// TIA Portal project "Hugo_Uriel_Travail_1" (V19)

(* hardware
DEVICE "HMI_1"  KTP700 Basic PN
   slot 0: "HMI_1"  KTP700 Basic PN  6AV2 123-2GB03-0AX0  17.0.0.0
   slot 1: "HMI_RT_1"  KTP700 Basic PN  6AV2 123-2GB03-0AX0  17.0.0.0
   slot 5: "HMI_1.IE_CP_1"  PROFINET Interface  17.0.0.0
      slot 1: "PROFINET Interface_1"  PROFINET Interface
         slot 1: "Port_1"  Port
DEVICE "S7-300/ET200M station_1"  S7-300 station
   slot 0: "Rail_0"  Rail  6ES7 390-1***0-0AA0
   slot 2: "PLC_1"  CPU 314C-2 PN/DP  6ES7 314-6EH04-0AB0  V3.3
      slot 2: "PROFINET interface_1"  PN-IO
         slot 1: "Port_1"  Port
         slot 2: "Port_2"  Port
      slot 5: "DI 24/DO 16_1"  DI24/DO16
      slot 6: "AI 5/AO 2_1"  AI5/AO2
      slot 7: "Count_1"  Counter
      slot 8: "Positioning_1"  Positioning
*)

// ===== PLC "PLC_1"  CPU 314C-2 PN/DP =====

VAR_GLOBAL   // PLC tag table "Default tag table"
   "Memoire pièce haute HMI" AT %M50.0 : Bool;
   "Memoire pièce basse HMI" AT %M50.1 : Bool;
   "Memoire pas de pièce HMI" AT %M50.2 : Bool;
   "Memoire B5" AT %M50.3 : Bool;
   "Memoire B6" AT %M50.4 : Bool;
   "HMI_M1" AT %M50.5 : Bool;
   "HMI_M2" AT %M50.6 : Bool;
   "HMI_1M1" AT %M50.7 : Bool;
   "HMI_2M1" AT %M51.0 : Bool;
END_VAR

VAR_GLOBAL   // PLC tag table "Variables Station Separating"
   "PART_AV" AT %I0.0 : Bool;   // Pièce Disponible
   "B2" AT %I0.1 : Bool;   // Présence pièce pour analyxe
   "B3" AT %I0.2 : Bool;   // Vérification profondeur pièce
   "B4" AT %I0.3 : Bool;   // Vérin rotatif rentré
   "B5" AT %I0.4 : Bool;   // Convoyeur 2 plein
   "B6" AT %I0.5 : Bool;   // Pièce en sortie de station
   "IP_FI_B" AT %I0.6 : Bool;   // Simulation station suivante libre
   "IP_FI" AT %I0.7 : Bool;   // Station suivante libre
   "BP Start" AT %I1.0 : Bool;   // NO Départ cycle
   "BP Stop" AT %I1.1 : Bool;   // NF Fin cycle
   "Selecteur Auto/Manu" AT %I1.2 : Bool;   // Choix mode fonctionnement
   "BP Reset" AT %I1.3 : Bool;   // Initialisation station
   "Emergency Stop" AT %I1.5 : Bool;   // Arrêt d'urgence (ponté)
   "M1" AT %Q0.0 : Bool;   // Convoyeur principal - Marche
   "M2" AT %Q0.1 : Bool;   // Convoyeur secondaire - Marche
   "1M1" AT %Q0.2 : Bool;   // Blocage pièce - sorti au repos
   "2M1" AT %Q0.3 : Bool;   // Aiguillage - convoyeur secondaire
   "IP_N_FO" AT %Q0.7 : Bool;   // Station occupée
   "LStart" AT %Q1.0 : Bool;   // Lampe BP Start
   "LReset" AT %Q1.1 : Bool;   // Lampe BP Reset
   "Q1" AT %Q1.2 : Bool;   // Voyant lumineux Gauche
   "Q2" AT %Q1.3 : Bool;   // Voyant lumineux Droite
   "B3 Analogique" AT %IW800 : Int;   // Profondeur Pièce
END_VAR

VAR_GLOBAL   // PLC tag table "Memoires"
   "FP0" AT %M30.0 : Bool;
   "FN0" AT %M31.0 : Bool;
   "FP1" AT %M30.1 : Bool;
   "FN1" AT %M31.1 : Bool;
   "Memoire_TP_Mesure" AT %M32.0 : Bool;
   "Memoire_TP_B5" AT %M32.1 : Bool;
   "RET_VAL" AT %MW10 : Word;
   "Sortie_Scale" AT %MD20 : Real;
   "Scale_bipolaire" AT %M33.0 : Bool;
   "FP2" AT %M30.2 : Bool;
   "FN2" AT %M31.2 : Bool;
   "FN3" AT %M31.3 : Bool;
   "Memoire_TP_B5_result" AT %M33.1 : Bool;
END_VAR

DATA_BLOCK "Tapis_roulant_DB_2"   // DB3
{ S7_Optimized_Access := 'FALSE' }
VERSION : 0.1
// stored: InstanceOfName Tapis_roulant_DB
"Tapis_roulant_DB"
BEGIN
END_DATA_BLOCK

DATA_BLOCK "Verrin_DB_Aiguillage"   // DB4
{ S7_Optimized_Access := 'FALSE' }
VERSION : 0.1
// stored: InstanceOfName Verrin_DB
"Verrin_DB"
BEGIN
END_DATA_BLOCK

DATA_BLOCK "Verrin_DB_blocage"   // DB5
{ S7_Optimized_Access := 'FALSE' }
VERSION : 0.1
// stored: InstanceOfName Verrin_DB
"Verrin_DB"
BEGIN
END_DATA_BLOCK

DATA_BLOCK "Data_block_memo"   // DB8
{ S7_Optimized_Access := 'FALSE' }
VERSION : 0.1
   VAR
      memo_convoyeur_1 : Bool;
      memo_convoyeur_2 : Bool;
      memo_verrin_aiguillage : Bool;
      memo_verrin_blocage : Bool;
      IN_Avancer_Tapis_1 : Bool;
      IN_Avancer_Tapis_2 : Bool;
      IN_Verrin_blocage : Bool;
      IN_Verrin_aiguillage : Bool;
      OUT_position_verrin_aiguillage : Bool;
      OUT_position_verrin_blocage : Bool;
      valeur_profondeur : Real;
      rent_val_capteur : Word;
      auto : Bool;
      manu : Bool;
      marche : Bool;
      arret : Bool;
      STATE : Int;
      profondeur : Bool;
   END_VAR
BEGIN
END_DATA_BLOCK

DATA_BLOCK "Tapis_roulant_DB_1"   // DB9
{ S7_Optimized_Access := 'FALSE' }
VERSION : 0.1
// stored: InstanceOfName Tapis_roulant_DB
"Tapis_roulant_DB"
BEGIN
END_DATA_BLOCK

DATA_BLOCK "Grafcet_DB"   // DB10
{ S7_Optimized_Access := 'FALSE' }
VERSION : 0.1
// stored: InstanceOfName Grafcet
"Grafcet"
BEGIN
END_DATA_BLOCK

FUNCTION_BLOCK "Verrin_DB"   // FB1, FBD
{ S7_Optimized_Access := 'FALSE' }
VERSION : 0.1
   VAR_INPUT
      Activation : Bool;
      Positon : Bool;
   END_VAR
   VAR_OUTPUT
      Marche : Bool;
      Position_retour : Bool;
   END_VAR
BEGIN

REGION Network 1
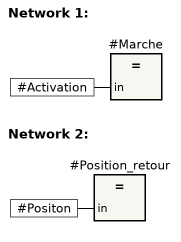
   #Marche := #Activation;
END_REGION

REGION Network 2
   #Position_retour := #Positon;
END_REGION
END_FUNCTION_BLOCK

FUNCTION_BLOCK "Tapis_roulant_DB"   // FB2, FBD
{ S7_Optimized_Access := 'FALSE' }
VERSION : 0.1
   VAR_INPUT
      Start_Avant : Bool;
   END_VAR
   VAR_OUTPUT
      Run : Bool;
   END_VAR
   VAR_TEMP
      moteur_tapis : Bool;
   END_VAR
BEGIN

REGION Network 1
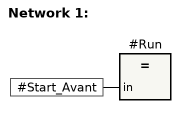
   #Run := #Start_Avant;
END_REGION
END_FUNCTION_BLOCK

FUNCTION_BLOCK "Grafcet"   // FB3, GRAPH
{ S7_Optimized_Access := 'FALSE' }
VERSION : 0.1
   VAR_INPUT
      OFF_SQ : Bool := false;   // Turn sequence off
      INIT_SQ : Bool := false;   // Set sequence to initial state
      ACK_EF : Bool := false;   // Acknowledge all errors and faults
      S_PREV : Bool := false;   // Output previous step in parameter S_NO
      S_NEXT : Bool := false;   // Indicate next step in parameter S_NO
      SW_AUTO : Bool := false;   // Automatic mode
      SW_TAP : Bool := false;   // Semiautomatic/switch with transition
      SW_TOP : Bool := false;   // Semiautomatic/ignore transition
      SW_MAN : Bool := false;   // Manual mode
      S_SEL : Int := 0;   // Select step to be output to S_NO
      S_ON : Bool := false;   // Activate step indicated in S_NO
      S_OFF : Bool := false;   // Disable step indicated in S_NO
      T_PUSH : Bool := false;   // Enable transition to switch in semi automatic mode
   END_VAR
   VAR_OUTPUT
      S_NO : Int := 0;   // Step number
      S_MORE : Bool := false;   // More steps are available and can be shown in S_NO
      S_ACTIVE : Bool := false;   // Step indicated in S_NO is active
      ERR_FLT : Bool := false;   // Interlock or supervision group error
      AUTO_ON : Bool := false;   // Automatic mode is active
      TAP_ON : Bool := false;   // Semiautomatic mode/step with transition enabled
      TOP_ON : Bool := false;   // Semiautomatic mode/ignore transition enabled
      MAN_ON : Bool := false;   // Manual mode is active
   END_VAR
   VAR
      SWITCH : Array[0..0] of DWord;
      SW_SQTS : Array[0..9] of Byte;
      SW_ADDR : Word := 16#A;
      G7T_0 : GraphTransition;
      G7S_0 : GraphStep;
      PRE_CRIT : Array[0..0] of DWord;
      POST_CRIT : Array[0..0] of DWord;
      TVX : Array[0..6] of Byte;
      TTX : Array[0..6] of Byte;
      TSX : Array[0..2] of Byte;
      S00X : Array[0..2] of Byte;
      SOFFX : Array[0..2] of Byte;
      SONX : Array[0..2] of Byte;
      SAX : Array[0..2] of Byte;
      SERRX : Array[0..10] of Byte;
      SMX : Array[0..10] of Byte;
      S0X : Array[0..10] of Byte;
      S1X : Array[0..10] of Byte;
      S_DISPLAY : Int;   // Internal display of output parameter S_NO
      S_SEL_OLD : Int;   // Previous value in S_SEL
      S_DISPIDX : Byte;   // Index of the step in S_NO
      T_DISPIDX : Byte;   // Index of the transition displayed in T_NO
      MOPEDGE : Struct
         AUTO : Bool := false;
         MAN : Bool := false;
         TAP : Bool := false;
         TOP : Bool := false;
         ACK_S : Bool := false;
         REG_S : Bool := false;
         T_PREV : Bool := false;
         T_NEXT : Bool := false;
         LOCK : Bool := false;
         SUP : Bool := false;
         ACKREQ : Bool := false;
         SSKIP : Bool := false;
         OFF : Bool := false;
         INIT : Bool := false;
         HALT : Bool := false;
         TMS_HALT : Bool := false;
         OPS_ZERO : Bool := false;
         SACT_DISP : Bool := false;
         SEF_DISP : Bool := false;
         SALL_DISP : Bool := false;
         S_PREV : Bool := false;
         S_NEXT : Bool := false;
         S_SELOK : Bool := false;
         S_ON : Bool := false;
         S_OFF : Bool := false;
         T_PUSH : Bool := false;
         REG : Bool := false;
         ACK : Bool := false;
         IL_PERM : Bool := false;
         T_PERM : Bool := false;
         ILP_MAN : Bool := false;
      END_STRUCT;
      MOP : Struct   // Mode
         AUTO : Bool := true;   // Status: automatic mode
         MAN : Bool := false;   // Status: manual mode
         TAP : Bool := false;   // Status: semi automatic/switch with transition
         TOP : Bool := false;   // Status: semi automatic/ignore transition
         ACK_S : Bool := false;   // Request: acknowledge step at parameter S_NO
         REG_S : Bool := false;   // Request: register step indicated in S_NO
         T_PREV : Bool := false;   // Request: output previous valid transition in T_NO
         T_NEXT : Bool := false;   // Request: output next valid transition in T_NO
         LOCK : Bool := true;   // Status: interlocks enabled
         SUP : Bool := true;   // Status: supervisions enabled
         ACKREQ : Bool := true;   // Status: acknowledgment required
         SSKIP : Bool := false;   // Status: "Skip steps" enabled
         OFF : Bool := false;   // Request: deactivate all steps
         INIT : Bool := true;   // Request: set sequence to initial state
         HALT : Bool := false;   // Status: sequence halted
         TMS_HALT : Bool := false;   // Status: all internal timers held
         OPS_ZERO : Bool := false;   // Status: set all operands processed with N, L, D instructions to 0
         SACT_DISP : Bool := true;   // Status: display active steps only
         SEF_DISP : Bool := false;   // Status: display only steps with errors and disrupted steps
         SALL_DISP : Bool := false;   // Status: display all steps
         S_PREV : Bool := false;   // Request: output previous step to S_NO
         S_NEXT : Bool := false;   // Request: Output next step at S_NO parameter
         S_SELOK : Bool := false;   // Request: output step number from S_SEL to S_NO
         S_ON : Bool := false;   // Request: activate step indicated in S_NO
         S_OFF : Bool := false;   // Request: deactivate step at parameter S_NO
         T_PUSH : Bool := false;   // Request: transition switching enabled
         REG : Bool := false;   // Request: register all interlock and supervision errors
         ACK : Bool := false;   // Request: acknowledge all interlock and supervision errors
         IL_PERM : Bool := false;   // Status: permanent processing of all interlocks
         T_PERM : Bool := false;   // Status: permanent processing of all transitions
         ILP_MAN : Bool := false;   // Status: permanent processing of all interlocks in manual mode
      END_STRUCT;
      TICKS : Struct   // Clock speeds
         DELTA : Time := T#0ms;   // Time difference between two cycles
         OLD : Time := T#0ms;   // 10 ms clock counter value in last cycle
         NEW : Time := T#0ms;   // 10 ms clock counter value in this cycle
      END_STRUCT;
      SQ_FLAGS : Struct   // Sequence bit memory
         ERR_FLT : Bool := false;   // Interlock and supervision group error
         ERROR : Bool := false;   // Interlock group error
         FAULT : Bool := false;   // Supervision group error
         RT_FAIL : Bool := false;   // Runtime error
         NO_SNO : Bool := false;   // Requested step number not found
         NF_OFL : Bool := false;   // Overflow: too many ON or OFF requests
         SA_OFL : Bool := false;   // Overflow: too many steps active
         TV_OFL : Bool := false;   // Overflow: too many valid transitions
         MSG_OFL : Bool := false;   // Overflow: not enough system resources for ALARM_S
         NO_SWI : Bool := false;   // Do not switch in this cycle
         CYC_OP : Bool := false;   // Cyclic execution of the sequence after initialization
         AS_MSG : Bool := true;   // Alarms during runtime enabled or disabled by instruction
         AS_SEND : Bool := false;   // Send alarms from WR_USMSG or only enter in diagnostics buffer
         SQ_BUSY : Bool := false;   // Internal edge bit memory for sequence processing
         SA_BUSY : Bool := false;   // Internal edge bit memory for sequence processing
         AS_SIG : Bool := false;   // Edge bit memory for alarms from Alarm_S and Alarm_SQ
      END_STRUCT;
      S_PTR : DWord := 16#6D0;
      S_PTR2 : DWord := 16#0;
      S_PTR3 : DWord := 16#1350;
      S_PTR4 : DWord := 16#12F0;
      T_PTR : DWord := 16#1290;
      C_AR2 : DWord := 16#0;
      M_FBDB : DWord := 16#30000;
      M_SNO : Word := 16#0;
      M_EVID : Word := 16#0;
      M_EVIL : C_Alarm_s;
      M_EVSV : C_Alarm_s;
      M_EV : DWord := 16#11D0;
      CRIT : Array[0..31] of Bool;
      S_START : Byte := 16#0;
      S_IDX : Byte := 16#0;
      S_INT : Int := 72;
      S_TMP : Byte := 16#0;
      T_START : Byte := 16#0;
      T_IDX : Byte := 16#0;
      T_TMP : Byte := 16#0;
      T_TMP2 : Byte := 16#00;
      TV_POT : Byte := 16#06;
      RETURN1 : Byte := 16#0;
      RETURN2 : Byte := 16#0;
      SINI : Array[0..2] of Byte;
      LSTT : Array[0..11] of Byte;
      ATAJ : Array[0..11] of Byte;
      ATAB : Array[0..11] of Byte;
      PSTT : Array[0..11] of Byte;
      NSTT : Array[0..11] of Byte;
      ASSJ : Array[0..9] of Byte;
      ASSB : Array[0..9] of Byte;
      PTTS : Array[0..9] of Byte;
      NTTS : Array[0..9] of Byte;
      PRE_CNT : Word := 16#1;
      POST_CNT : Word := 16#1;
      ADR_COND : Word := 16#0;
      MAX_TVAL : Byte := 16#5;
      MAX_SACT : Byte := 16#1;
      MAX_CRIT : Byte := 16#4;
      T_CNT : Byte := 16#B;
      SUP_CNT : Byte := 16#0;
      LOCK_CNT : Byte := 16#0;
      S_CNT : Byte := 16#9;
      SQ_CNT : Byte := 16#1;
      PRS_INPAR : DWord := 16#E000FEC8;
      PRS_OUTPAR : DWord := 16#E000800F;
      GC_FLAGS : Struct
         T_MACH : Byte := 16#EB;
         COND_ED : Byte := 16#E3;
         W_LEVEL : Byte := 16#D5;
         FB_IF : Byte := 16#FA;
         AS_MSG : Word := 16#404;
         SSB : Word := 16#108;
         DILG : Word := 16#35E;
         ADDR_T0 : Word := 16#1A;
         CRIT_AVAIL : Bool := false;
         SSKIP_AVAIL : Bool := true;
         SSKIP_ON : Bool := false;
         ACK_REQ : Bool := true;
         SYNC_AVAIL : Bool := true;
         ILP_MAN : Bool := false;
         SWM_LOCKED : Bool := false;
         SAVE_SW : Bool := true;
      END_STRUCT;
      G7_FBMARK : Byte := 16#3C;
      G7_RELEASE : Byte := 16#3C;
      G7_ID2 : Byte := 16#37;
      G7_ID1 : Byte := 16#47;
   END_VAR
   // SW_SQTS[0] := 16#5;
   // SW_SQTS[5] := 16#2;
   // SW_SQTS[4] := 16#1;
   // SW_SQTS[3] := 16#1;
   // SW_SQTS[6] := 16#2;
   // SW_SQTS[7] := 16#3;
   // SW_SQTS[8] := 16#3;
   // SW_SQTS[9] := 16#4;
   // TVX[0] := 16#1;
   // TTX[0] := 16#1;
   // TSX[0] := 16#1;
   // S00X[0] := 16#1;
   // SOFFX[0] := 16#1;
   // SONX[0] := 16#1;
   // SAX[0] := 16#1;
   // SERRX[0] := 16#1;
   // SMX[0] := 16#1;
   // S0X[0] := 16#1;
   // S1X[0] := 16#1;
   // SINI[0] := 16#2;
   // SINI[1] := 16#1;
   // SINI[2] := 0;
   // LSTT[0] := 0;
   // LSTT[1] := 0;
   // LSTT[2] := 0;
   // LSTT[3] := 0;
   // LSTT[4] := 0;
   // LSTT[5] := 0;
   // LSTT[6] := 0;
   // LSTT[7] := 16#3;
   // LSTT[8] := 0;
   // LSTT[9] := 0;
   // LSTT[10] := 16#3;
   // LSTT[11] := 16#2;
   // ATAJ[0] := 0;
   // ATAJ[1] := 16#1;
   // ATAJ[2] := 16#2;
   // ATAJ[3] := 16#3;
   // ATAJ[4] := 16#4;
   // ATAJ[5] := 16#5;
   // ATAJ[6] := 16#6;
   // ATAJ[7] := 16#7;
   // ATAJ[8] := 16#8;
   // ATAJ[9] := 16#9;
   // ATAJ[10] := 16#A;
   // ATAJ[11] := 16#B;
   // ATAB[0] := 0;
   // ATAB[1] := 16#1;
   // ATAB[2] := 16#3;
   // ATAB[3] := 16#2;
   // ATAB[4] := 16#4;
   // ATAB[5] := 16#8;
   // ATAB[6] := 16#6;
   // ATAB[7] := 16#7;
   // ATAB[8] := 16#5;
   // ATAB[9] := 16#9;
   // ATAB[10] := 16#A;
   // ATAB[11] := 16#B;
   // PSTT[0] := 0;
   // PSTT[1] := 16#1;
   // PSTT[2] := 16#2;
   // PSTT[3] := 16#2;
   // PSTT[4] := 16#3;
   // PSTT[5] := 16#4;
   // PSTT[6] := 16#5;
   // PSTT[7] := 16#6;
   // PSTT[8] := 16#4;
   // PSTT[9] := 16#7;
   // PSTT[10] := 16#8;
   // PSTT[11] := 16#9;
   // NSTT[0] := 16#1;
   // NSTT[1] := 16#2;
   // NSTT[2] := 16#3;
   // NSTT[3] := 16#9;
   // NSTT[4] := 16#4;
   // NSTT[5] := 16#5;
   // NSTT[6] := 16#6;
   // NSTT[7] := 16#3;
   // NSTT[8] := 16#7;
   // NSTT[9] := 16#8;
   // NSTT[10] := 16#3;
   // NSTT[11] := 16#2;
   // ASSJ[0] := 0;
   // ASSJ[1] := 16#1;
   // ASSJ[2] := 16#2;
   // ASSJ[3] := 16#3;
   // ASSJ[4] := 16#4;
   // ASSJ[5] := 16#5;
   // ASSJ[6] := 16#6;
   // ASSJ[7] := 16#7;
   // ASSJ[8] := 16#8;
   // ASSJ[9] := 16#9;
   // ASSB[0] := 0;
   // ASSB[1] := 16#1;
   // ASSB[2] := 16#2;
   // ASSB[3] := 16#3;
   // ASSB[4] := 16#4;
   // ASSB[5] := 16#5;
   // ASSB[6] := 16#6;
   // ASSB[7] := 16#7;
   // ASSB[8] := 16#8;
   // ASSB[9] := 16#9;
   // PTTS[0] := 0;
   // PTTS[2] := 16#1;
   // PTTS[3] := 16#2;
   // PTTS[4] := 16#4;
   // PTTS[5] := 16#5;
   // PTTS[6] := 16#6;
   // PTTS[7] := 16#8;
   // PTTS[8] := 16#9;
   // PTTS[9] := 16#3;
   // NTTS[0] := 0;
   // NTTS[1] := 16#1;
   // NTTS[2] := 16#2;
   // NTTS[3] := 16#4;
   // NTTS[4] := 16#5;
   // NTTS[5] := 16#6;
   // NTTS[6] := 16#7;
   // NTTS[7] := 16#9;
   // NTTS[8] := 16#A;
   // NTTS[9] := 16#B;
BEGIN
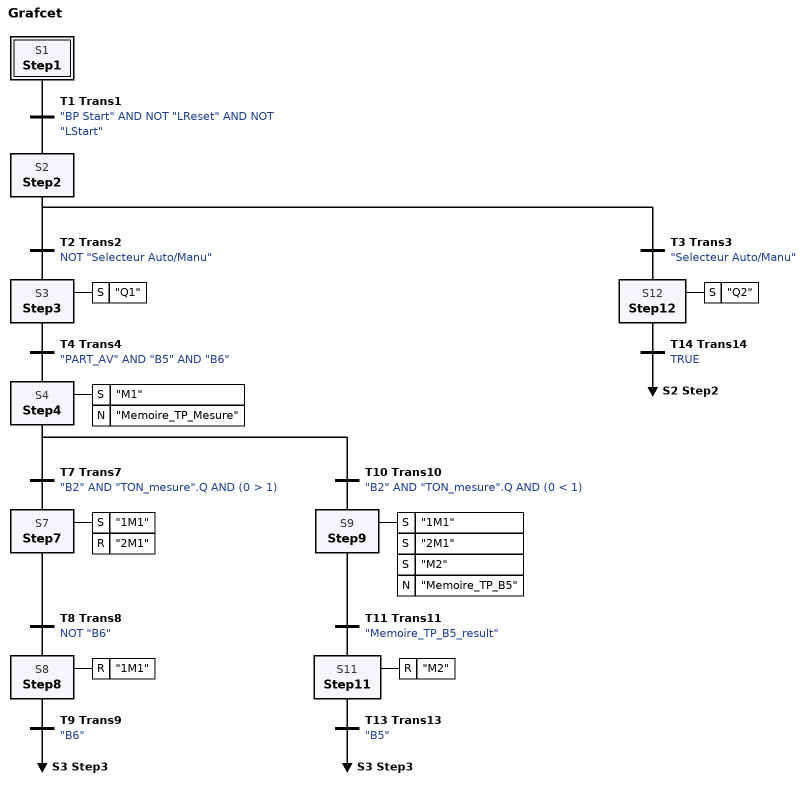
   // sequencer 1
   INITIAL_STEP Step1:   // S1
   END_STEP
   TRANSITION Trans1 FROM Step1 TO Step2   // T1
      := "BP Start" AND NOT "LReset" AND NOT "LStart";
   END_TRANSITION
   STEP Step2:   // S2
   END_STEP
   TRANSITION Trans2 FROM Step2 TO Step3   // T2
      := NOT "Selecteur Auto/Manu";
   END_TRANSITION
   TRANSITION Trans3 FROM Step2 TO Step12   // T3
      := "Selecteur Auto/Manu";
   END_TRANSITION
   STEP Step3:   // S3
              S    "Q1"
   END_STEP
   TRANSITION Trans4 FROM Step3 TO Step4   // T4
      := "PART_AV" AND "B5" AND "B6";
   END_TRANSITION
   STEP Step4:   // S4
              S    "M1"
              N    "Memoire_TP_Mesure"
   END_STEP
   TRANSITION Trans7 FROM Step4 TO Step7   // T7
      := "B2" AND "TON_mesure".Q AND (0 > 1);
   END_TRANSITION
   TRANSITION Trans10 FROM Step4 TO Step9   // T10
      := "B2" AND "TON_mesure".Q AND (0 < 1);
   END_TRANSITION
   STEP Step7:   // S7
              S    "1M1"
              R    "2M1"
   END_STEP
   TRANSITION Trans8 FROM Step7 TO Step8   // T8
      := NOT "B6";
   END_TRANSITION
   STEP Step8:   // S8
              R    "1M1"
   END_STEP
   TRANSITION Trans9 FROM Step8 TO Step3   // T9, jump
      := "B6";
   END_TRANSITION
   STEP Step9:   // S9
              S    "1M1"
              S    "2M1"
              S    "M2"
              N    "Memoire_TP_B5"
   END_STEP
   TRANSITION Trans11 FROM Step9 TO Step11   // T11
      := "Memoire_TP_B5_result";
   END_TRANSITION
   STEP Step11:   // S11
              R    "M2"
   END_STEP
   TRANSITION Trans13 FROM Step11 TO Step3   // T13, jump
      := "B5";
   END_TRANSITION
   STEP Step12:   // S12
              S    "Q2"
   END_STEP
   TRANSITION Trans14 FROM Step12 TO Step2   // T14, jump
      := TRUE;
   END_TRANSITION
END_FUNCTION_BLOCK

FUNCTION "Mesure hauteur HMI" : Void   // FC1, LAD
{ S7_Optimized_Access := 'FALSE' }
VERSION : 0.1
// Petit bloc FC qui permetl'affichage du type de pièce au niveau de la mesure pour l'HMI
BEGIN

REGION Network 1: Pièce haute
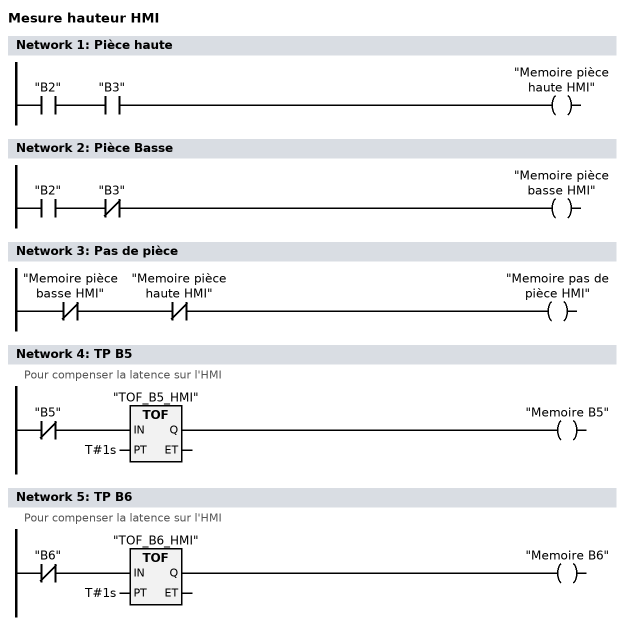
   RUNG wire#powerrail
      Contact( "B2" )
      Contact( "B3" )
      Coil( "Memoire pièce haute HMI" )
   END_RUNG
   // the same network as SCL:
   "Memoire pièce haute HMI" := "B2" AND "B3";
END_REGION

REGION Network 2: Pièce Basse
   RUNG wire#powerrail
      Contact( "B2" )
      I_Contact( "B3" )
      Coil( "Memoire pièce basse HMI" )
   END_RUNG
   // the same network as SCL:
   "Memoire pièce basse HMI" := "B2" AND NOT "B3";
END_REGION

REGION Network 3: Pas de pièce
   RUNG wire#powerrail
      I_Contact( "Memoire pièce basse HMI" )
      I_Contact( "Memoire pièce haute HMI" )
      Coil( "Memoire pas de pièce HMI" )
   END_RUNG
   // the same network as SCL:
   "Memoire pas de pièce HMI" := NOT "Memoire pièce basse HMI" AND NOT "Memoire pièce haute HMI";
END_REGION

REGION Network 4: TP B5
   // Pour compenser la latence sur l'HMI
   "TOF_B5_HMI".TOF(IN := NOT "B5", PT := T#1s);
   "Memoire B5" := "TOF_B5_HMI".Q;
END_REGION

REGION Network 5: TP B6
   // Pour compenser la latence sur l'HMI
   "TOF_B6_HMI".TOF(IN := NOT "B6", PT := T#1s);
   "Memoire B6" := "TOF_B6_HMI".Q;
END_REGION
END_FUNCTION

FUNCTION "Mode_auto" : Void   // FC2, FBD
{ S7_Optimized_Access := 'FALSE' }
VERSION : 0.1
   VAR_TEMP
      false : Bool;
      State : Int;
      Mode_auto : Bool;
   END_VAR
   VAR_TEMP   // added for the SCL form of the ladder/FBD networks
      _w1 : Bool;
   END_VAR
BEGIN

REGION Network 1
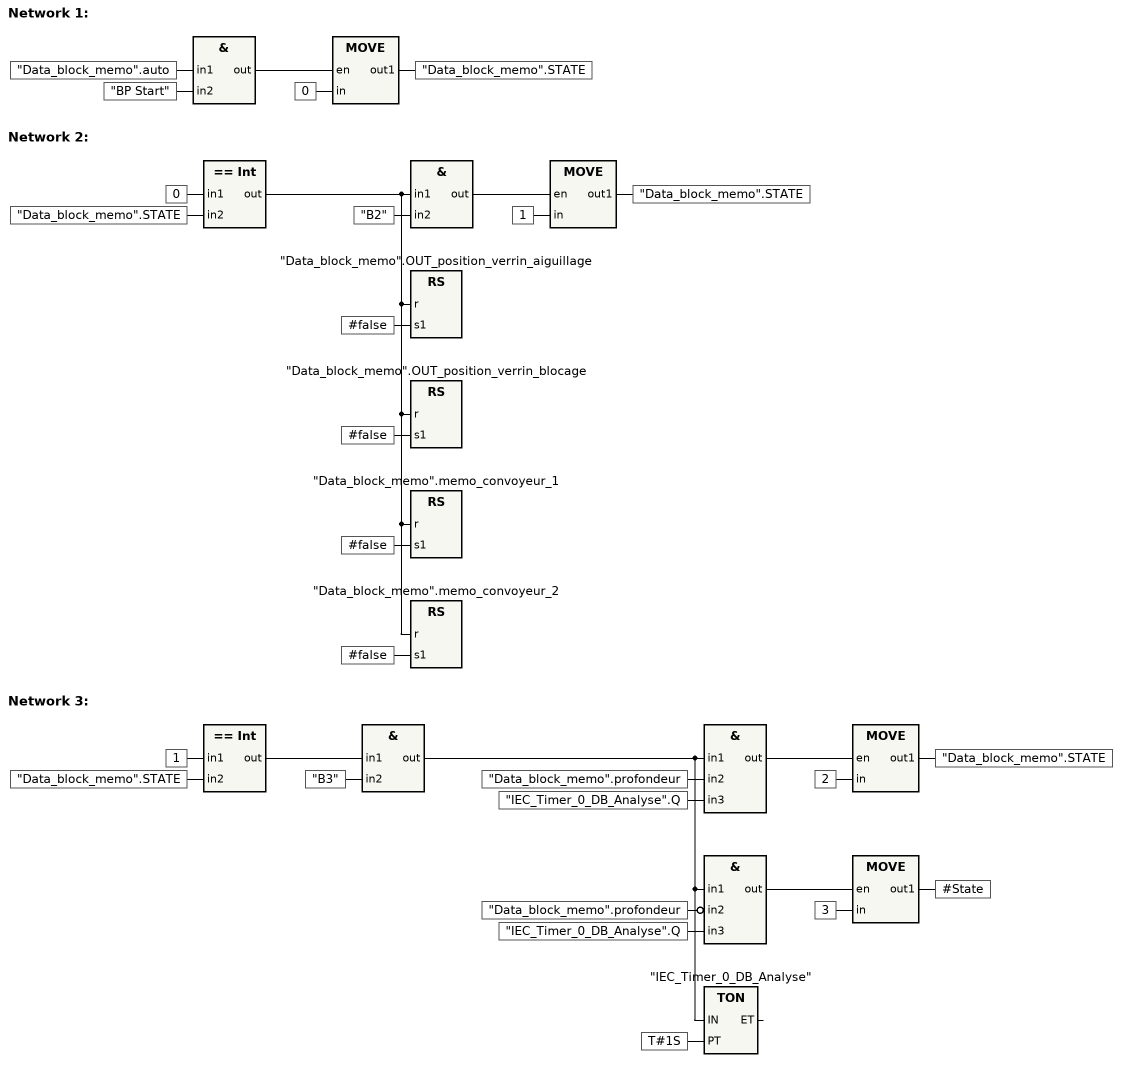
   IF "Data_block_memo".auto AND "BP Start" THEN "Data_block_memo".STATE := 0; END_IF;
END_REGION

REGION Network 2
   #_w1 := 0 = "Data_block_memo".STATE;
   IF #_w1 AND "B2" THEN "Data_block_memo".STATE := 1; END_IF;
   IF #_w1 THEN
       "Data_block_memo".OUT_position_verrin_aiguillage := FALSE;   // RS flip-flop
   END_IF;
   IF #false THEN "Data_block_memo".OUT_position_verrin_aiguillage := TRUE; END_IF;
   IF #_w1 THEN
       "Data_block_memo".OUT_position_verrin_blocage := FALSE;   // RS flip-flop
   END_IF;
   IF #false THEN "Data_block_memo".OUT_position_verrin_blocage := TRUE; END_IF;
   IF #_w1 THEN
       "Data_block_memo".memo_convoyeur_1 := FALSE;   // RS flip-flop
   END_IF;
   IF #false THEN "Data_block_memo".memo_convoyeur_1 := TRUE; END_IF;
   IF #_w1 THEN
       "Data_block_memo".memo_convoyeur_2 := FALSE;   // RS flip-flop
   END_IF;
   IF #false THEN "Data_block_memo".memo_convoyeur_2 := TRUE; END_IF;
END_REGION

REGION Network 3
   #_w1 := (1 = "Data_block_memo".STATE) AND "B3";
   IF #_w1 AND "Data_block_memo".profondeur AND "IEC_Timer_0_DB_Analyse".Q THEN
       "Data_block_memo".STATE := 2;
   END_IF;
   IF #_w1 AND NOT "Data_block_memo".profondeur AND "IEC_Timer_0_DB_Analyse".Q THEN #State := 3; END_IF;
   "IEC_Timer_0_DB_Analyse".TON(IN := #_w1, PT := T#1S);
END_REGION

REGION Network 4
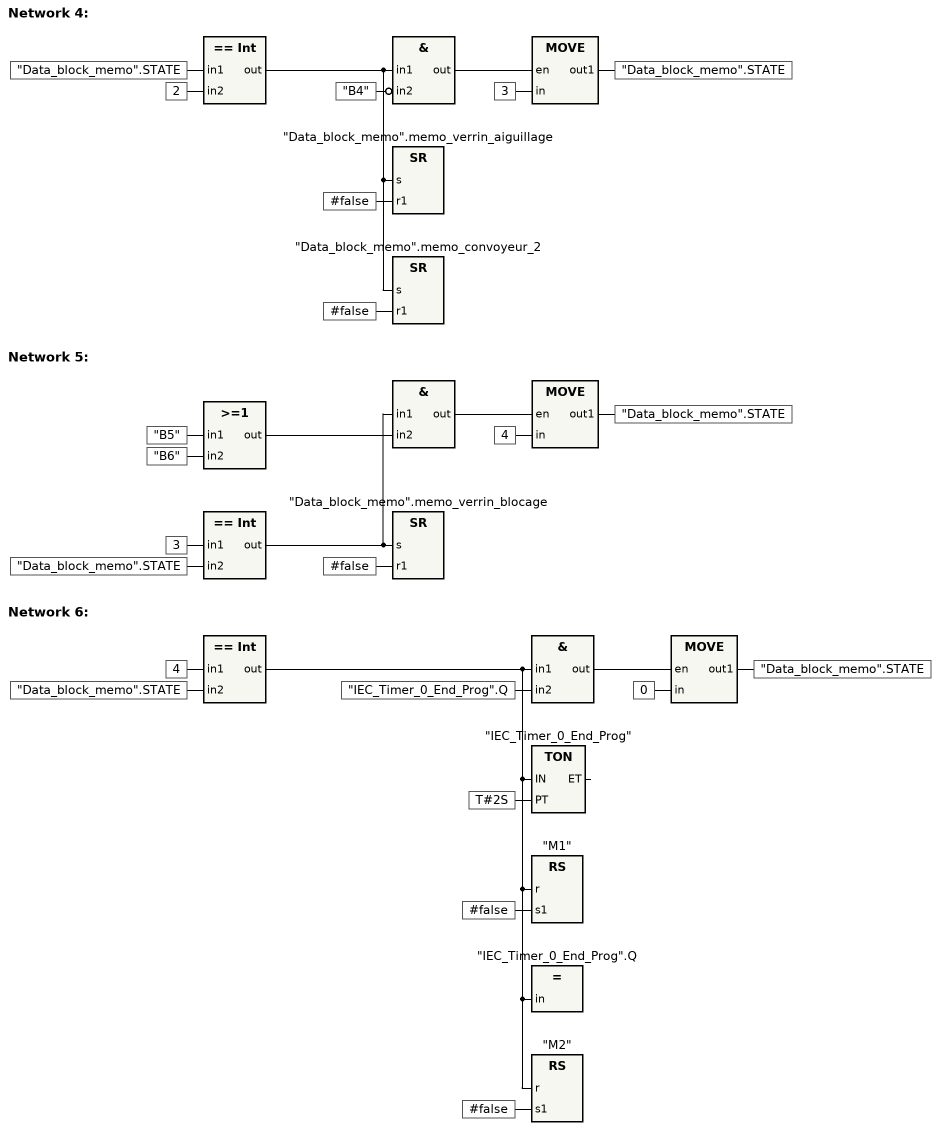
   #_w1 := "Data_block_memo".STATE = 2;
   IF #_w1 AND NOT "B4" THEN "Data_block_memo".STATE := 3; END_IF;
   IF #_w1 THEN
       "Data_block_memo".memo_verrin_aiguillage := TRUE;   // SR flip-flop
   END_IF;
   IF #false THEN "Data_block_memo".memo_verrin_aiguillage := FALSE; END_IF;
   IF #_w1 THEN
       "Data_block_memo".memo_convoyeur_2 := TRUE;   // SR flip-flop
   END_IF;
   IF #false THEN "Data_block_memo".memo_convoyeur_2 := FALSE; END_IF;
END_REGION

REGION Network 5
   #_w1 := 3 = "Data_block_memo".STATE;
   IF #_w1 AND ("B5" OR "B6") THEN "Data_block_memo".STATE := 4; END_IF;
   IF #_w1 THEN
       "Data_block_memo".memo_verrin_blocage := TRUE;   // SR flip-flop
   END_IF;
   IF #false THEN "Data_block_memo".memo_verrin_blocage := FALSE; END_IF;
END_REGION

REGION Network 6
   #_w1 := 4 = "Data_block_memo".STATE;
   IF #_w1 AND "IEC_Timer_0_End_Prog".Q THEN "Data_block_memo".STATE := 0; END_IF;
   "IEC_Timer_0_End_Prog".TON(IN := #_w1, PT := T#2S);
   IF #_w1 THEN
       "M1" := FALSE;   // RS flip-flop
   END_IF;
   IF #false THEN "M1" := TRUE; END_IF;
   "IEC_Timer_0_End_Prog".Q := #_w1;
   IF #_w1 THEN
       "M2" := FALSE;   // RS flip-flop
   END_IF;
   IF #false THEN "M2" := TRUE; END_IF;
END_REGION
END_FUNCTION

FUNCTION "Lecteure/Ecriture_analogique" : Void   // FC3, FBD
{ S7_Optimized_Access := 'FALSE' }
VERSION : 0.1
   VAR_INPUT
      Valeur_IN : Int;
   END_VAR
   VAR_OUTPUT
      Valeur_OUT : Real;
      Ret_val_1 : Word;
   END_VAR
   VAR_TEMP
      Mem_Valeur_out : Real;
   END_VAR
   VAR CONSTANT
      Bipolar : Bool;
   END_VAR
BEGIN

REGION Network 1
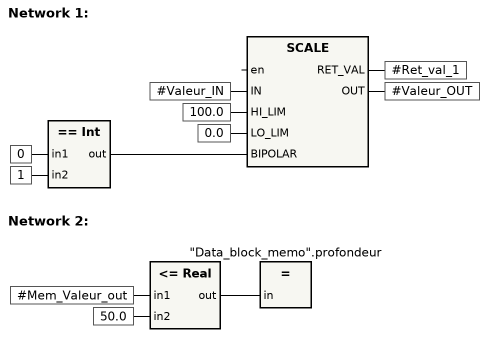
   #Ret_val_1 := SCALE(IN := #Valeur_IN, HI_LIM := 100.0, LO_LIM := 0.0, BIPOLAR := 0 = 1, OUT => #Valeur_OUT);
END_REGION

REGION Network 2
   "Data_block_memo".profondeur := #Mem_Valeur_out <= 50.0;
END_REGION
END_FUNCTION

FUNCTION "Mode-focntionnement" : Void   // FC4, FBD
{ S7_Optimized_Access := 'FALSE' }
VERSION : 0.1
   VAR_INPUT
      "Auto/Manu" : Bool;
      Start : Bool;
      Stop : Bool;
      Reset : Bool;
   END_VAR
   VAR_OUTPUT
      Auto_out : Bool;
      Manu_out : Bool;
      Mode_marche : Bool;
      Mode_arret : Bool;
   END_VAR
   VAR_TEMP
      marche_mem : Bool;
      P_trig_changement : Bool;
      P_trig_changement_1 : Bool;
      false : Bool;
      Arret_mem : Bool;
   END_VAR
BEGIN

REGION Network 1
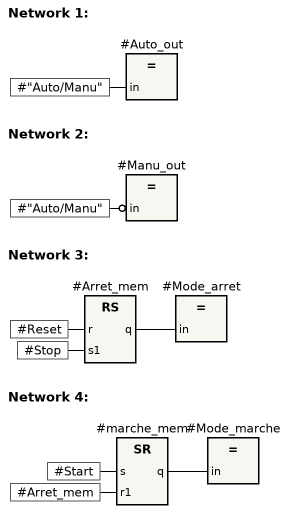
   #Auto_out := #"Auto/Manu";
END_REGION

REGION Network 2
   #Manu_out := NOT #"Auto/Manu";
END_REGION

REGION Network 3
   IF #Reset THEN
       #Arret_mem := FALSE;   // RS flip-flop
   END_IF;
   IF #Stop THEN #Arret_mem := TRUE; END_IF;
   #Mode_arret := #Arret_mem;
END_REGION

REGION Network 4
   IF #Start THEN
       #marche_mem := TRUE;   // SR flip-flop
   END_IF;
   IF #Arret_mem THEN #marche_mem := FALSE; END_IF;
   #Mode_marche := #marche_mem;
END_REGION
END_FUNCTION

FUNCTION "mode_manu" : Void   // FC5, FBD
{ S7_Optimized_Access := 'FALSE' }
VERSION : 0.1
BEGIN

REGION Network 1: Tapis 1
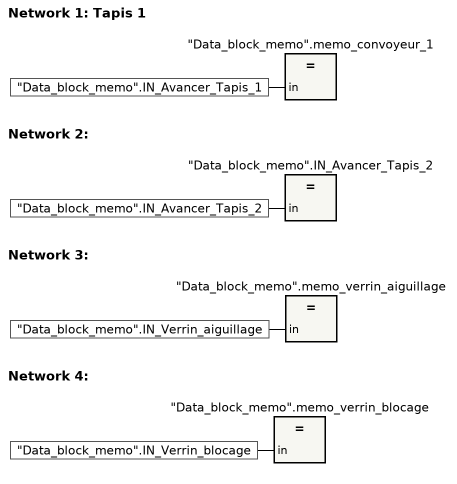
   "Data_block_memo".memo_convoyeur_1 := "Data_block_memo".IN_Avancer_Tapis_1;
END_REGION

REGION Network 2
   "Data_block_memo".IN_Avancer_Tapis_2 := "Data_block_memo".IN_Avancer_Tapis_2;
END_REGION

REGION Network 3
   "Data_block_memo".memo_verrin_aiguillage := "Data_block_memo".IN_Verrin_aiguillage;
END_REGION

REGION Network 4
   "Data_block_memo".memo_verrin_blocage := "Data_block_memo".IN_Verrin_blocage;
END_REGION
END_FUNCTION

FUNCTION "Alimentation" : Void   // FC6, LAD
{ S7_Optimized_Access := 'FALSE' }
VERSION : 0.1
   VAR_TEMP   // added for the SCL form of the ladder/FBD networks
      _w1 : Bool;
      _w2 : Bool;
   END_VAR
BEGIN

REGION Network 1: Gestion Start
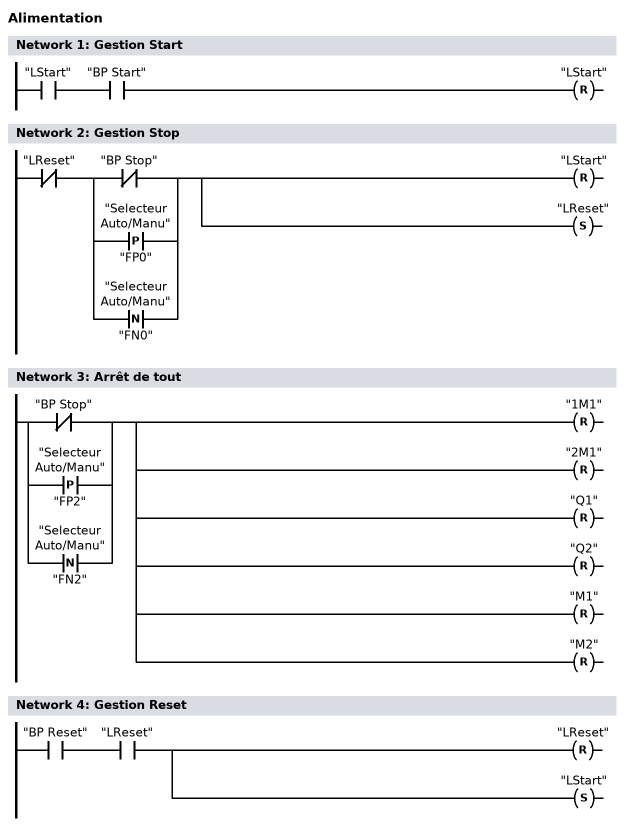
   RUNG wire#powerrail
      Contact( "LStart" )
      Contact( "BP Start" )
      R_Coil( "LStart" )
   END_RUNG
   // the same network as SCL:
   IF "LStart" AND "BP Start" THEN "LStart" := FALSE; END_IF;
END_REGION

REGION Network 2: Gestion Stop
   RUNG wire#powerrail
      I_Contact( "LReset" )
      wire#w1
      I_Contact( "BP Stop" )
      wire#w2
      R_Coil( "LStart" )
   END_RUNG
   RUNG wire#w1
      P_Contact(operand := "Selecteur Auto/Manu", bit := "FP0")
   END_RUNG wire#w2
   RUNG wire#w1
      N_Contact(operand := "Selecteur Auto/Manu", bit := "FN0")
   END_RUNG wire#w2
   RUNG wire#w2
      S_Coil( "LReset" )
   END_RUNG
   // the same network as SCL:
   #_w1 := NOT "LReset" AND "Selecteur Auto/Manu" AND NOT "FP0";   // rising edge of "Selecteur Auto/Manu"
   "FP0" := "Selecteur Auto/Manu";
   #_w2 := NOT "LReset" AND NOT "Selecteur Auto/Manu" AND "FN0";   // falling edge of "Selecteur Auto/Manu"
   "FN0" := "Selecteur Auto/Manu";
   IF (NOT "LReset" AND NOT "BP Stop") OR #_w1 OR #_w2 THEN
       "LStart" := FALSE;
       "LReset" := TRUE;
   END_IF;
END_REGION

REGION Network 3: Arrêt de tout
   RUNG wire#powerrail
      I_Contact( "BP Stop" )
      wire#w1
      R_Coil( "1M1" )
   END_RUNG
   RUNG wire#powerrail
      P_Contact(operand := "Selecteur Auto/Manu", bit := "FP2")
   END_RUNG wire#w1
   RUNG wire#powerrail
      N_Contact(operand := "Selecteur Auto/Manu", bit := "FN2")
   END_RUNG wire#w1
   RUNG wire#w1
      R_Coil( "2M1" )
   END_RUNG
   RUNG wire#w1
      R_Coil( "Q1" )
   END_RUNG
   RUNG wire#w1
      R_Coil( "Q2" )
   END_RUNG
   RUNG wire#w1
      R_Coil( "M1" )
   END_RUNG
   RUNG wire#w1
      R_Coil( "M2" )
   END_RUNG
   // the same network as SCL:
   #_w1 := "Selecteur Auto/Manu" AND NOT "FP2";   // rising edge of "Selecteur Auto/Manu"
   "FP2" := "Selecteur Auto/Manu";
   #_w2 := NOT "Selecteur Auto/Manu" AND "FN2";   // falling edge of "Selecteur Auto/Manu"
   "FN2" := "Selecteur Auto/Manu";
   IF NOT "BP Stop" OR #_w1 OR #_w2 THEN
       "1M1" := FALSE;
       "2M1" := FALSE;
       "Q1" := FALSE;
       "Q2" := FALSE;
       "M1" := FALSE;
       "M2" := FALSE;
   END_IF;
END_REGION

REGION Network 4: Gestion Reset
   RUNG wire#powerrail
      Contact( "BP Reset" )
      Contact( "LReset" )
      wire#w1
      R_Coil( "LReset" )
   END_RUNG
   RUNG wire#w1
      S_Coil( "LStart" )
   END_RUNG
   // the same network as SCL:
   #_w1 := "BP Reset" AND "LReset";
   IF #_w1 THEN
       "LReset" := FALSE;
       "LStart" := TRUE;
   END_IF;
END_REGION
END_FUNCTION

FUNCTION "Tempo Grafcet" : Void   // FC7, LAD
{ S7_Optimized_Access := 'FALSE' }
VERSION : 0.1
   VAR_TEMP   // added for the SCL form of the ladder/FBD networks
      _w1 : Bool;
   END_VAR
BEGIN

REGION Network 1
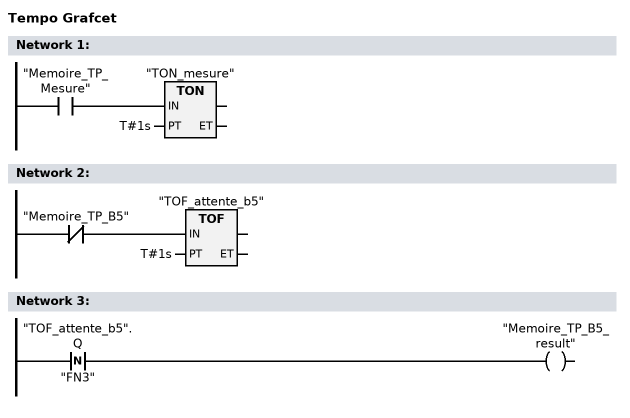
   "TON_mesure".TON(IN := "Memoire_TP_Mesure", PT := T#1s);
END_REGION

REGION Network 2
   "TOF_attente_b5".TOF(IN := NOT "Memoire_TP_B5", PT := T#1s);
END_REGION

REGION Network 3
   RUNG wire#powerrail
      N_Contact(operand := "TOF_attente_b5".Q, bit := "FN3")
      Coil( "Memoire_TP_B5_result" )
   END_RUNG
   // the same network as SCL:
   #_w1 := NOT "TOF_attente_b5".Q AND "FN3";   // falling edge of "TOF_attente_b5".Q
   "FN3" := "TOF_attente_b5".Q;
   "Memoire_TP_B5_result" := #_w1;
END_REGION
END_FUNCTION

ORGANIZATION_BLOCK "Main"   // OB1, LAD
TITLE = "Main Program Sweep (Cycle)"
{ S7_Optimized_Access := 'FALSE' }
VERSION : 0.1
   VAR_TEMP
      OB1_EV_CLASS : Byte;   // Bits 0-3 = 1 (Coming event), Bits 4-7 = 1 (Event class 1)
      OB1_SCAN_1 : Byte;   // 1 (Cold restart scan 1 of OB 1), 3 (Scan 2-n of OB 1)
      OB1_PRIORITY : Byte;   // Priority of OB Execution
      OB1_OB_NUMBR : Byte;   // 1 (Organization block 1, OB1)
      OB1_RESERVED_1 : Byte;   // Reserved for system
      OB1_RESERVED_2 : Byte;   // Reserved for system
      OB1_PREV_CYCLE : Int;   // Cycle time of previous OB1 scan (milliseconds)
      OB1_MIN_CYCLE : Int;   // Minimum cycle time of OB1 (milliseconds)
      OB1_MAX_CYCLE : Int;   // Maximum cycle time of OB1 (milliseconds)
      OB1_DATE_TIME : Date_And_Time;   // Date and time OB1 started
   END_VAR
   VAR_TEMP   // added for the SCL form of the ladder/FBD networks
      _w1 : Bool;
      _w2 : Bool;
   END_VAR
BEGIN

REGION Network 1: Gestion Alimentation
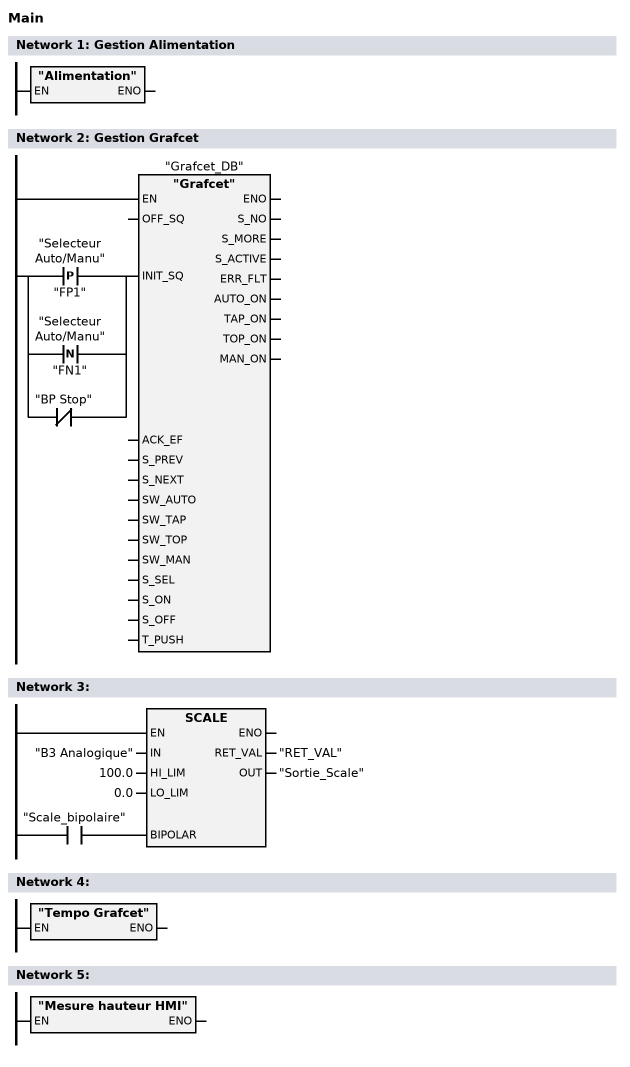
   RUNG wire#powerrail
      "Alimentation"()
   END_RUNG
   // the same network as SCL:
   "Alimentation"();
END_REGION

REGION Network 2: Gestion Grafcet
   RUNG wire#powerrail
      "Grafcet_DB"(INIT_SQ := wire#w1, OFF_SQ :=, ACK_EF :=, S_PREV :=, S_NEXT :=, SW_AUTO :=, SW_TAP :=, SW_TOP :=, SW_MAN :=, S_SEL :=, S_ON :=, S_OFF :=, T_PUSH :=, S_NO =>, S_MORE =>, S_ACTIVE =>, ERR_FLT =>, AUTO_ON =>, TAP_ON =>, TOP_ON =>, MAN_ON =>)
   END_RUNG
   RUNG wire#powerrail
      P_Contact(operand := "Selecteur Auto/Manu", bit := "FP1")
   END_RUNG wire#w1
   RUNG wire#powerrail
      N_Contact(operand := "Selecteur Auto/Manu", bit := "FN1")
   END_RUNG wire#w1
   RUNG wire#powerrail
      I_Contact( "BP Stop" )
   END_RUNG wire#w1
   // the same network as SCL:
   #_w1 := "Selecteur Auto/Manu" AND NOT "FP1";   // rising edge of "Selecteur Auto/Manu"
   "FP1" := "Selecteur Auto/Manu";
   #_w2 := NOT "Selecteur Auto/Manu" AND "FN1";   // falling edge of "Selecteur Auto/Manu"
   "FN1" := "Selecteur Auto/Manu";
   "Grafcet_DB"(INIT_SQ := #_w1 OR #_w2 OR NOT "BP Stop");   // "Grafcet"
END_REGION

REGION Network 3
   "RET_VAL" := SCALE(IN := "B3 Analogique",
                      HI_LIM := 100.0,
                      LO_LIM := 0.0,
                      BIPOLAR := "Scale_bipolaire",
                      OUT => "Sortie_Scale");
END_REGION

REGION Network 4
   RUNG wire#powerrail
      "Tempo Grafcet"()
   END_RUNG
   // the same network as SCL:
   "Tempo Grafcet"();
END_REGION

REGION Network 5
   RUNG wire#powerrail
      "Mesure hauteur HMI"()
   END_RUNG
   // the same network as SCL:
   "Mesure hauteur HMI"();
END_REGION
END_ORGANIZATION_BLOCK

ORGANIZATION_BLOCK "COMPLETE RESTART"   // OB100, LAD
TITLE = "Complete Restart"
{ S7_Optimized_Access := 'FALSE' }
VERSION : 0.1
   VAR_TEMP
      OB100_EV_CLASS : Byte;   // 16#13, Event class 1, Entering event state, Event logged in diagnostic buffer
      OB100_STRTUP : Byte;   // 16#81/82/83/84 Method of startup
      OB100_PRIORITY : Byte;   // Priority of OB Execution
      OB100_OB_NUMBR : Byte;   // 100 (Organization block 100, OB100)
      OB100_RESERVED_1 : Byte;   // Reserved for system
      OB100_RESERVED_2 : Byte;   // Reserved for system
      OB100_STOP : Word;   // Event that caused CPU to stop (16#4xxx)
      OB100_STRT_INFO : DWord;   // Information on how system started
      OB100_DATE_TIME : Date_And_Time;   // Date and time OB100 started
   END_VAR
BEGIN

REGION Network 1: Lampe BP Reset
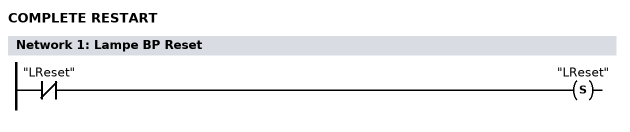
   RUNG wire#powerrail
      I_Contact( "LReset" )
      S_Coil( "LReset" )
   END_RUNG
   // the same network as SCL:
   IF NOT "LReset" THEN "LReset" := TRUE; END_IF;
END_REGION
END_ORGANIZATION_BLOCK

(* ===== HMI "HMI_RT_1" =====
system functions are stored by id; their names below are inferred from use
connection "HMI_Connection_1": ETHERNET, SIMATIC S7 300/400 MPI

HMI tags "Default tag table"
   "Tag_ScreenNumber" : UInt, internal
   "Nom_utilisateur" : WString[254], internal
   "M1" : Bool = PLC M1 AT %Q0.0, 1 s
   "M2" : Bool = PLC M2 AT %Q0.1, 1 s
   "1M1" : Bool = PLC 1M1 AT %Q0.2, 1 s
   "2M1" : Bool = PLC 2M1 AT %Q0.3, 1 s
   "PART_AV" : Bool = PLC PART_AV AT %I0.0, 1 s
   "B2" : Bool = PLC B2 AT %I0.1, 1 s
   "B3" : Bool = PLC B3 AT %I0.2, 1 s
   "B4" : Bool = PLC B4 AT %I0.3, 1 s
   "B5" : Bool = PLC "Memoire B5" AT %M50.3, 1 s
   "B6" : Bool = PLC "Memoire B6" AT %M50.4, 1 s
   "Pièce haute" : Bool = PLC "Memoire pièce haute HMI" AT %M50.0, 1 s
   "Pièce basse" : Bool = PLC "Memoire pièce basse HMI" AT %M50.1, 1 s
   "Pas de pièce" : Bool = PLC "Memoire pas de pièce HMI" AT %M50.2, 1 s

Template "Template_1" 800x480
   Button "Exit" at 714,429 size 71x50; TextOff 'Exit'; PictureOff "ExitRuntime_KTP700_Basic_PN_TR"; PictureOn "ExitRuntime_KTP700_Basic_PN_TR"
      on Release: StopRuntime(0)
   Button "Template_Button" at 614,429 size 71x50; TextOff 'Text'
   Button "Template_Button_1" at 514,410 size 71x69; TextOff 'Text'; PictureOff "Logo utilisateur"; Authorization "User administration"
      on Release: ActivateScreen("Page Utilisateurs", 0)
   Button "Template_Button_2" at 414,410 size 71x69; TextOff 'Text'; PictureOff "Logo historique"
      on Release: ActivateScreen("Page Historique", 0)
   Button "Template_Button_3" at 314,410 size 71x69; TextOff 'Text'; PictureOff "Logo Automatique"
      on Release: ActivateScreen("Page Mode Automatique", 0)
   Button "Template_Button_4" at 214,410 size 71x69; TextOff 'Text'; PictureOff "Logo Manuel"; Authorization "Monitor"
      on Release: ActivateScreen("Page Mode Manuel", 0)
   Button "Alarms" at 114,429 size 71x50; TextOff 'Alarms'; PictureOff "AlarmDisplay_KTP700_Basic_PN_TR"; PictureOn "AlarmDisplay_KTP700_Basic_PN_TR"
      on Release: function_ef3f5d25("Alarm window_Unacknowledged", -1)
   Button "Start screen" at 14,429 size 71x50; TextOff 'Start screen'; PictureOff "NavigateHome_KTP700_Basic_PN_TR"; PictureOn "NavigateHome_KTP700_Basic_PN_TR"
      on Release: ActivateScreen("Page d'accueil", 0)
   DateTimeField "HmiScreenItemData" at 695,25 size 105x25
   DateTimeField "HmiScreenItemData_1" at 695,0 size 105x25
   TextField "Template_Text field_1" at 277,5 size 196x23; Text 'Connecté en tant que :'
   IOField "I/O field_1" at 473,3 size 113x33; FormatPattern ????????????????????????????????????????????????????????????????????????????????
      ProcessValue <- "Nom_utilisateur"

screen "Page d'accueil" 800x480, template "Template_1"
   on GenerateScreen: SetTag("Tag_ScreenNumber", 1)
   TextField "HmiScreenItemData" at 154,293 size 198x25; Text 'Travail 1'
   TextField "HmiScreenItemData_1" at 154,332 size 195x25; Text 'Par Uriel et Hugo'
   GraphicView "Graphic view_1" at 154,43 size 195x226; Picture "Logo_HENALLUX-removebg-preview"
   Button "Button_1" at 545,171 size 96x32; TextOff 'Login'
      on Activate: function_a2a04561()
   Button "Button_2" at 545,230 size 96x32; TextOff 'Logout'
      on Activate: function_f23ef4c9()

screen "Page Historique" 800x480, template "Template_1"
   TextField "Text field_1" at 11,5 size 136x34; Text 'Historique'

screen "Page Utilisateurs" 800x480, template "Template_1"
   TextField "Text field_1" at 11,5 size 150x34; Text 'Utilisateurs'
   Button "Button_1" at 269,63 size 96x32; TextOff 'Login'
      on Activate: function_a2a04561()
   Button "Button_2" at 404,63 size 96x32; TextOff 'Logout'
      on Activate: function_f23ef4c9()
   UserView "User view_1" at 0,128 size 798x240

screen "Page Mode Automatique" 800x480, template "Template_1"
   TextField "Text field_1" at 11,5 size 242x34; Text 'Mode Automatique'
   Line "Line_1" at 374,198 size 51x0
      Visibility <- "B5"
   Line "Line_2" at 565,246 size 0x52
      Visibility <- "B6"
   Line "Line_3" at 361,319 size 95x0
      Visibility <- "2M1"
   Line "Line_4" at 359,252 size 71x66
      Visibility <- "2M1"
   Line "Line_5" at 236,245 size 8x11
      Visibility <- "PART_AV"
   Line "Line_6" at 228,244 size 8x13
      Visibility <- "PART_AV"
   Line "Line_7" at 236,245 size 0x14
      Visibility <- "PART_AV"
   Line "Line_8" at 285,283 size 8x13
      Visibility <- "B2"
   Line "Line_9" at 294,282 size 0x14
      Visibility <- "B2"
   Line "Line_10" at 294,284 size 9x14
      Visibility <- "B2"
   Line "Line_11" at 324,270 size 0x28
      Visibility <- "1M1"
   Line "Line_12" at 246,272 size 26x0
      Visibility <- "M1"
   Line "Line_13" at 263,272 size 9x8
      Visibility <- "M1"
   Line "Line_14" at 264,265 size 8x7
      Visibility <- "M1"
   Line "Line_15" at 484,272 size 26x0
      Visibility <- "M1"
   Line "Line_16" at 501,272 size 9x8
      Visibility <- "M1"
   Line "Line_17" at 502,265 size 8x7
      Visibility <- "M1"
   Line "Line_18" at 401,162 size 0x23
      Visibility <- "M2"
   Line "Line_19" at 401,162 size 6x9
      Visibility <- "M2"
   Line "Line_20" at 395,162 size 6x9
      Visibility <- "M2"
   TextField "Text field_2" at 217,153 size 107x23; Text 'Pas de pièce'
      Visibility <- "Pas de pièce"
   TextField "Text field_3" at 217,153 size 101x23; Text 'Pièce haute'
      Visibility <- "Pièce haute"
   TextField "Text field_4" at 217,153 size 100x23; Text 'Pièce basse'
      Visibility <- "Pièce basse"

screen "Page Mode Manuel" 800x480, template "Template_1"
   TextField "Text field_1" at 11,5 size 172x34; Text 'Mode Manuel'
   Line "Line_1" at 517,136 size 51x0
      Visibility <- "B5"
   Switch "Switch_1" at 547,308 size 213x83; CaptionText 'Switch'; TextOff 'Tapis Principal'; TextOn 'Tapis Secondaire'
      on SwitchOn: SetBit("2M1")
      on SwitchOff: ResetBit("2M1")
   Switch "Switch_2" at 292,308 size 213x83; CaptionText 'Switch'; TextOff 'Pièce Bloquée'; TextOn 'Passage libre'
      on SwitchOn: SetBit("1M1")
      on SwitchOff: ResetBit("1M1")
   Switch "Switch_3" at 39,308 size 213x83; CaptionText 'Switch'; TextOff 'M2 Stop'; TextOn 'M2 Marche'
      on SwitchOn: SetBit("M2")
      on SwitchOff: ResetBit("M2")
   Line "Line_2" at 708,184 size 0x52
      Visibility <- "B6"
   Line "Line_3" at 504,257 size 95x0
      Visibility <- "2M1"
   Line "Line_4" at 502,190 size 71x66
      Visibility <- "2M1"
   Line "Line_5" at 379,183 size 8x11
      Visibility <- "PART_AV"
   Line "Line_6" at 371,182 size 8x13
      Visibility <- "PART_AV"
   Line "Line_7" at 379,183 size 0x14
      Visibility <- "PART_AV"
   Line "Line_8" at 428,221 size 8x13
      Visibility <- "B2"
   Line "Line_9" at 437,220 size 0x14
      Visibility <- "B2"
   Line "Line_10" at 437,222 size 9x14
      Visibility <- "B2"
   Line "Line_11" at 467,208 size 0x28
      Visibility <- "1M1"
   Line "Line_12" at 389,210 size 26x0
      Visibility <- "M1"
   Line "Line_13" at 406,210 size 9x8
      Visibility <- "M1"
   Line "Line_14" at 407,203 size 8x7
      Visibility <- "M1"
   Line "Line_15" at 627,210 size 26x0
      Visibility <- "M1"
   Line "Line_16" at 644,210 size 9x8
      Visibility <- "M1"
   Line "Line_17" at 645,203 size 8x7
      Visibility <- "M1"
   Line "Line_18" at 544,100 size 0x23
      Visibility <- "M2"
   Line "Line_19" at 544,100 size 6x9
      Visibility <- "M2"
   Line "Line_20" at 538,100 size 6x9
      Visibility <- "M2"
   Switch "Switch_4" at 40,183 size 213x83; CaptionText 'Switch'; TextOff 'M1 Stop'; TextOn 'M1 Marche'
      on SwitchOn: SetBit("M1")
      on SwitchOff: ResetBit("M1")
   TextField "Text field_2" at 360,91 size 107x23; Text 'Pas de pièce'
      Visibility <- "Pas de pièce"
   TextField "Text field_3" at 360,91 size 101x23; Text 'Pièce haute'
      Visibility <- "Pièce haute"
   TextField "Text field_4" at 360,91 size 100x23; Text 'Pièce basse'
      Visibility <- "Pièce basse"

scheduled task "Task_1"
   on Action: function_f41c6f6c("Nom_utilisateur")
*)